(* PLC project Prototype, Beckhoff Automation GmbH TwinCAT PLC Control 3.5.13.21 *)
(* stored: creationDateTime 2023-12-06T16:09:30.7727106, modificationDateTime 2023-12-06T16:09:30.7795414 *)

INTERFACE ITF_Shape
METHOD Clone : ITF_Shape
VAR_INPUT
END_VAR
END_METHOD
METHOD Draw
VAR_INPUT
END_VAR
END_METHOD
END_INTERFACE

{attribute 'enable_dynamic_creation'}
FUNCTION_BLOCK Circle IMPLEMENTS ITF_Shape
VAR_INPUT
	radius: INT;
END_VAR
VAR_OUTPUT
END_VAR
VAR
END_VAR

                  
                

METHOD  Clone : ITF_Shape
VAR_INPUT
END_VAR
VAR_STAT
 pClone : POINTER TO Circle;	
END_VAR
                        pClone := __NEW(Circle);
pClone^.radius := radius;
Clone := pClone^;
__DELETE(pClone);

                      
END_METHOD

METHOD Draw

VAR
	str : STRING;
END_VAR
                        str := TO_STRING(radius);

ADSLOGSTR(msgCtrlMask :=ADSLOG_MSGTYPE_HINT, msgFmtStr :='Draw circle with radius: %s', strArg := str);
                      
END_METHOD
END_FUNCTION_BLOCK

{attribute 'enable_dynamic_creation'}
FUNCTION_BLOCK Rectangle IMPLEMENTS ITF_Shape
VAR_INPUT
	width: INT;
    height: INT;
END_VAR
VAR_OUTPUT
END_VAR
VAR
END_VAR

                  
                

METHOD Clone : ITF_Shape
VAR_INPUT
END_VAR
VAR_STAT
	clonedRectangle: Rectangle;
END_VAR
                        clonedRectangle.width := width;
clonedRectangle.height := height;

Clone := clonedRectangle;
                      
END_METHOD

METHOD Draw

VAR
	str_width : STRING;
	str_height: STRING;
	str : STRING;
END_VAR
                        
str_width  := CONCAT(STR1:= 'width: ', STR2:=  TO_STRING(width));
str_height := CONCAT(STR1:= 'height: ', STR2:=  TO_STRING(height));
str :=  CONCAT(STR1:= str_width, STR2:=  str_height);

ADSLOGSTR(msgCtrlMask :=ADSLOG_MSGTYPE_HINT, msgFmtStr :='Draw Rectangle with:  %s', strArg := str);
                      
END_METHOD
END_FUNCTION_BLOCK

PROGRAM MAIN
VAR
    originalRectangle: Rectangle;
    clonedRectangle: ITF_Shape;
	
    originalCircle: Circle;
    clonedCircle: ITF_Shape;
	
	bRequest : BOOL;

END_VAR

                  // https://refactoring.guru/design-patterns/prototype

// Recuerda que el patrón Prototipo permite crear nuevos objetos clonando un objeto existente, evitando así la necesidad de crear nuevas instancias desde cero.


IF bRequest THEN
	
	originalRectangle.width := 10;
	originalRectangle.height := 5;
	originalRectangle.Draw();
	clonedRectangle := originalRectangle.clone();
	clonedRectangle.Draw();
	
	originalCircle.radius := 7;
	originalCircle.Draw();
	clonedCircle := originalCircle.clone();
	clonedCircle.Draw();
		
	bRequest := FALSE;
	

END_IF
                
END_PROGRAM

CONFIGURATION Application
  RESOURCE Prototype ON PLC
    TASK PlcTask(INTERVAL := T#0ms, PRIORITY := 20);
    PROGRAM MAIN WITH PlcTask : MAIN;
  END_RESOURCE
END_CONFIGURATION
